
FUNCTION CB_bool_to_word : WORD

TITLE = ' Convert a boolean into an word '
VERSION : '1.0'
AUTHOR  : CB
NAME    : boToWord
FAMILY  : TNI

VAR_INPUT
    IN : BOOL;
END_VAR

VAR_TEMP

END_VAR

BEGIN

CB_bool_to_word := INT_TO_WORD(BOOL_TO_INT(IN));

END_FUNCTION
